GLOBALCONSTANTS logiBUS_2_CAN_DI (* logiBUS_DI constants *)
  (* Standard: 61499-1; Description: Copyright (c) 2024 HR Agrartechnik GmbH This program and the accompanying materials are made available under the terms of the Eclipse Public License 2.0 which is available at https://www.eclipse.org/legal/epl-2.0/ SPDX-License-Identifier: EPL-2.0 *)
  (* Version 1.0, 2024-01-25, Franz Höpfinger, HR Agrartechnik GmbH *)
  VAR_GLOBAL CONSTANT
    Input_I1 : logiBUS_2_CAN_DI_S := (Pin := 1);
    Input_I2 : logiBUS_2_CAN_DI_S := (Pin := 2);
    Invalid : logiBUS_2_CAN_DI_S := (Pin := 255);
  END_VAR
END_GLOBALCONSTANTS
